TYPE ST_HardSettings_ParallelOperation :
STRUCT
	b_MasterSlaveEnabled				: BOOL;
	b_UnitIsMaster						: BOOL;
	b_ShutdownOnCommError				: BOOL;
	b_EffiencyMode						: BOOL; //Control inverter start/stop depending on load. Make load share algorithm.
	r_VoltageDroop						: REAL;
	r_FrequencyDroop					: REAL;
END_STRUCT
END_TYPE

(* stored: Version 1.1.0.1, ProductVersion 3.1.4026.18
   DUT ST_HardSettings_ParallelOperation: Id {a3124d2c-4233-404c-b81c-a3733390e728} *)
